PROGRAM OP10_ROBO
VAR
	I_OP10A_6000_6007						: BYTE_AS_BIT;	
	I_OP10A_6008_6015                       : BYTE_AS_BIT;
	I_OP10A_6016_6023                       : BYTE_AS_BIT;
	I_OP10A_6024_6031                       : BYTE_AS_BIT;
	I_OP10A_6032_6039                       : BYTE_AS_BIT;
	I_OP10A_6040_6047                       : BYTE_AS_BIT;
	I_OP10A_6048_6055                       : BYTE_AS_BIT;
	I_OP10A_6056_6063                       : BYTE_AS_BIT;
	O_OP10A_6000_6007						: BIT_AS_BYTE;
	O_OP10A_6008_6015						: BIT_AS_BYTE;
	O_OP10A_6016_6023						: BIT_AS_BYTE;
	O_OP10A_6024_6031						: BIT_AS_BYTE;
	O_OP10A_6032_6039						: BIT_AS_BYTE;
	O_OP10A_6040_6047						: BIT_AS_BYTE;
	O_OP10A_6048_6055						: BIT_AS_BYTE;
	O_OP10A_6056_6063						: BIT_AS_BYTE;

	I_OP10B_6000_6007						: BYTE_AS_BIT;	
	I_OP10B_6008_6015                       : BYTE_AS_BIT;
	I_OP10B_6016_6023                       : BYTE_AS_BIT;
	I_OP10B_6024_6031                       : BYTE_AS_BIT;
	I_OP10B_6032_6039                       : BYTE_AS_BIT;
	I_OP10B_6040_6047                       : BYTE_AS_BIT;
	I_OP10B_6048_6055                       : BYTE_AS_BIT;
	I_OP10B_6056_6063                       : BYTE_AS_BIT;
	O_OP10B_6032_6039						: BIT_AS_BYTE;
	O_OP10B_6040_6047						: BIT_AS_BYTE;
	O_OP10B_6048_6055						: BIT_AS_BYTE;
	O_OP10B_6056_6063						: BIT_AS_BYTE;
	O_OP10B_6000_6007						: BIT_AS_BYTE;
	O_OP10B_6008_6015						: BIT_AS_BYTE;
	O_OP10B_6016_6023						: BIT_AS_BYTE;
	O_OP10B_6024_6031						: BIT_AS_BYTE;

	OP10A_IP_ROBO_6000_6007  AT %I*			: USINT;
	OP10A_IP_ROBO_6008_6015  AT %I*			: USINT;
	OP10A_IP_ROBO_6016_6023  AT %I*			: USINT;
	OP10A_IP_ROBO_6024_6031  AT %I*			: USINT;
	OP10A_IP_ROBO_6032_6039  AT %I*			: USINT;
	OP10A_IP_ROBO_6040_6047  AT %I*			: USINT;	
	OP10A_IP_ROBO_6048_6055  AT %I*			: USINT;	
	OP10A_IP_ROBO_6056_6063  AT %I*			: USINT;	
	OP10A_OP_ROBO_6000_6007  AT %Q*			: USINT;
	OP10A_OP_ROBO_6008_6015  AT %Q*			: USINT;
	OP10A_OP_ROBO_6016_6023  AT %Q*			: USINT;
	OP10A_OP_ROBO_6024_6031  AT %Q*			: USINT;
	OP10A_OP_ROBO_6032_6039  AT %Q*			: USINT;
	OP10A_OP_ROBO_6040_6047  AT %Q*			: USINT;	
	OP10A_OP_ROBO_6048_6055  AT %Q*			: USINT;	
	OP10A_OP_ROBO_6056_6063  AT %Q*			: USINT;

	OP10B_IP_ROBO_6000_6007  AT %I*			: USINT;
	OP10B_IP_ROBO_6008_6015  AT %I*			: USINT;
	OP10B_IP_ROBO_6016_6023  AT %I*			: USINT;
	OP10B_IP_ROBO_6024_6031  AT %I*			: USINT;
	OP10B_IP_ROBO_6032_6039  AT %I*			: USINT;
	OP10B_IP_ROBO_6040_6047  AT %I*			: USINT;	
	OP10B_IP_ROBO_6048_6055  AT %I*			: USINT;	
	OP10B_IP_ROBO_6056_6063  AT %I*			: USINT;
	OP10B_OP_ROBO_6000_6007  AT %Q*			: USINT;
	OP10B_OP_ROBO_6008_6015  AT %Q*			: USINT;
	OP10B_OP_ROBO_6016_6023  AT %Q*			: USINT;
	OP10B_OP_ROBO_6024_6031  AT %Q*			: USINT;
	OP10B_OP_ROBO_6032_6039  AT %Q*			: USINT;
	OP10B_OP_ROBO_6040_6047  AT %Q*			: USINT;	
	OP10B_OP_ROBO_6048_6055  AT %Q*			: USINT;	
	OP10B_OP_ROBO_6056_6063  AT %Q*			: USINT;	


	


END_VAR

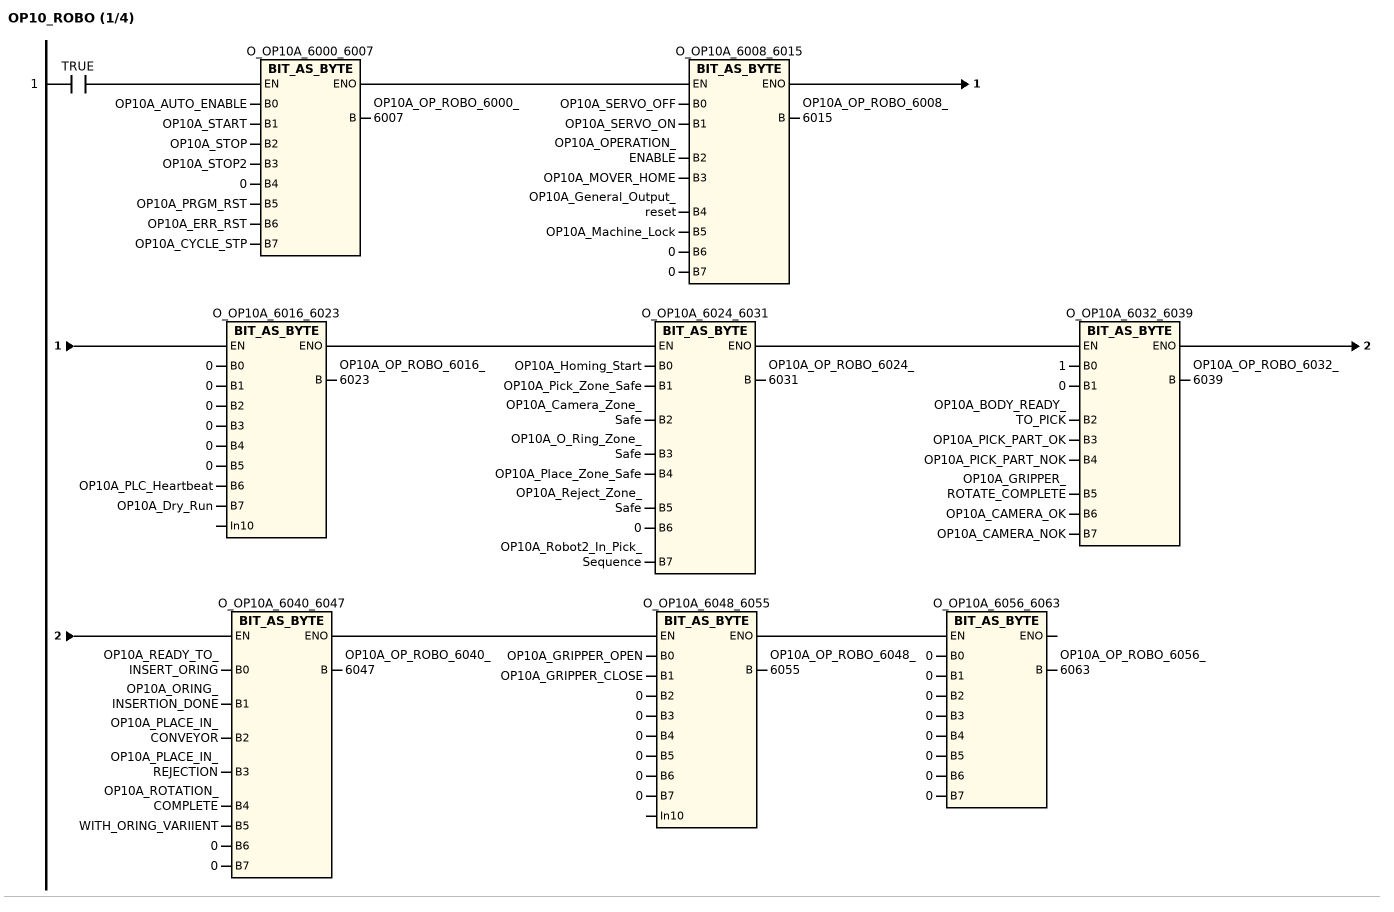
// NETWORK 1
O_OP10A_6000_6007(
    B0 := OP10A_AUTO_ENABLE,
    B1 := OP10A_START,
    B2 := OP10A_STOP,
    B3 := OP10A_STOP2,
    B4 := 0,
    B5 := OP10A_PRGM_RST,
    B6 := OP10A_ERR_RST,
    B7 := OP10A_CYCLE_STP,
    B => OP10A_OP_ROBO_6000_6007); // BIT_AS_BYTE
O_OP10A_6008_6015(
    B0 := OP10A_SERVO_OFF,
    B1 := OP10A_SERVO_ON,
    B2 := OP10A_OPERATION_ENABLE,
    B3 := OP10A_MOVER_HOME,
    B4 := OP10A_General_Output_reset,
    B5 := OP10A_Machine_Lock,
    B6 := 0,
    B7 := 0,
    B => OP10A_OP_ROBO_6008_6015); // BIT_AS_BYTE
O_OP10A_6016_6023(
    B0 := 0,
    B1 := 0,
    B2 := 0,
    B3 := 0,
    B4 := 0,
    B5 := 0,
    B6 := OP10A_PLC_Heartbeat,
    B7 := OP10A_Dry_Run,
    B => OP10A_OP_ROBO_6016_6023); // BIT_AS_BYTE
O_OP10A_6024_6031(
    B0 := OP10A_Homing_Start,
    B1 := OP10A_Pick_Zone_Safe,
    B2 := OP10A_Camera_Zone_Safe,
    B3 := OP10A_O_Ring_Zone_Safe,
    B4 := OP10A_Place_Zone_Safe,
    B5 := OP10A_Reject_Zone_Safe,
    B6 := 0,
    B7 := OP10A_Robot2_In_Pick_Sequence,
    B => OP10A_OP_ROBO_6024_6031); // BIT_AS_BYTE
O_OP10A_6032_6039(
    B0 := 1,
    B1 := 0,
    B2 := OP10A_BODY_READY_TO_PICK,
    B3 := OP10A_PICK_PART_OK,
    B4 := OP10A_PICK_PART_NOK,
    B5 := OP10A_GRIPPER_ROTATE_COMPLETE,
    B6 := OP10A_CAMERA_OK,
    B7 := OP10A_CAMERA_NOK,
    B => OP10A_OP_ROBO_6032_6039); // BIT_AS_BYTE
O_OP10A_6040_6047(
    B0 := OP10A_READY_TO_INSERT_ORING,
    B1 := OP10A_ORING_INSERTION_DONE,
    B2 := OP10A_PLACE_IN_CONVEYOR,
    B3 := OP10A_PLACE_IN_REJECTION,
    B4 := OP10A_ROTATION_COMPLETE,
    B5 := WITH_ORING_VARIIENT,
    B6 := 0,
    B7 := 0,
    B => OP10A_OP_ROBO_6040_6047); // BIT_AS_BYTE
O_OP10A_6048_6055(
    B0 := OP10A_GRIPPER_OPEN,
    B1 := OP10A_GRIPPER_CLOSE,
    B2 := 0,
    B3 := 0,
    B4 := 0,
    B5 := 0,
    B6 := 0,
    B7 := 0,
    B => OP10A_OP_ROBO_6048_6055); // BIT_AS_BYTE
O_OP10A_6056_6063(
    B0 := 0,
    B1 := 0,
    B2 := 0,
    B3 := 0,
    B4 := 0,
    B5 := 0,
    B6 := 0,
    B7 := 0,
    B => OP10A_OP_ROBO_6056_6063); // BIT_AS_BYTE

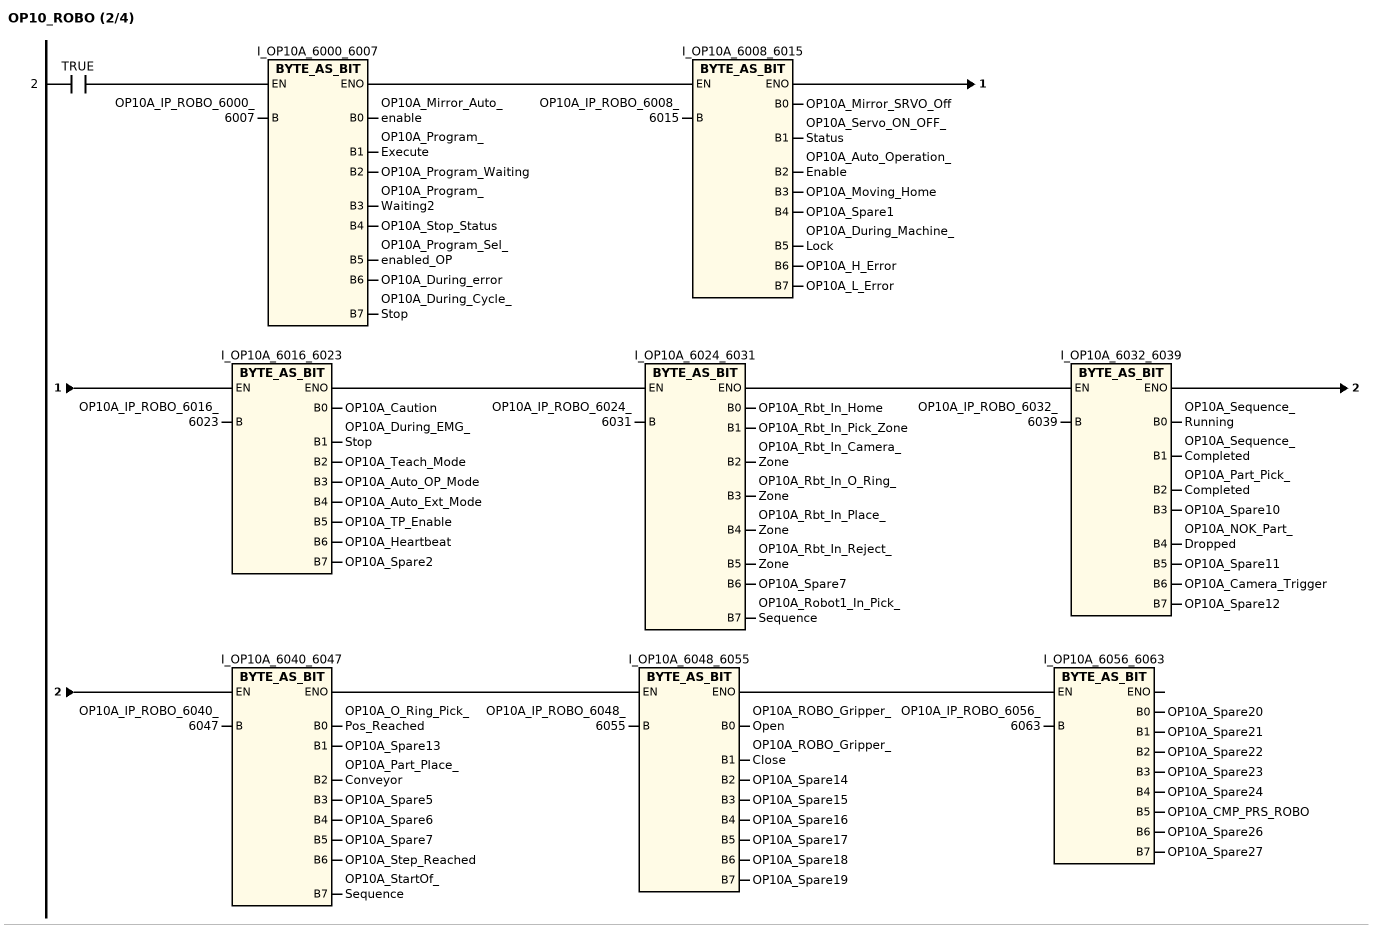
// NETWORK 2
I_OP10A_6000_6007(
    B := OP10A_IP_ROBO_6000_6007,
    B0 => OP10A_Mirror_Auto_enable,
    B1 => OP10A_Program_Execute,
    B2 => OP10A_Program_Waiting,
    B3 => OP10A_Program_Waiting2,
    B4 => OP10A_Stop_Status,
    B5 => OP10A_Program_Sel_enabled_OP,
    B6 => OP10A_During_error,
    B7 => OP10A_During_Cycle_Stop); // BYTE_AS_BIT
I_OP10A_6008_6015(
    B := OP10A_IP_ROBO_6008_6015,
    B0 => OP10A_Mirror_SRVO_Off,
    B1 => OP10A_Servo_ON_OFF_Status,
    B2 => OP10A_Auto_Operation_Enable,
    B3 => OP10A_Moving_Home,
    B4 => OP10A_Spare1,
    B5 => OP10A_During_Machine_Lock,
    B6 => OP10A_H_Error,
    B7 => OP10A_L_Error); // BYTE_AS_BIT
I_OP10A_6016_6023(
    B := OP10A_IP_ROBO_6016_6023,
    B0 => OP10A_Caution,
    B1 => OP10A_During_EMG_Stop,
    B2 => OP10A_Teach_Mode,
    B3 => OP10A_Auto_OP_Mode,
    B4 => OP10A_Auto_Ext_Mode,
    B5 => OP10A_TP_Enable,
    B6 => OP10A_Heartbeat,
    B7 => OP10A_Spare2); // BYTE_AS_BIT
I_OP10A_6024_6031(
    B := OP10A_IP_ROBO_6024_6031,
    B0 => OP10A_Rbt_In_Home,
    B1 => OP10A_Rbt_In_Pick_Zone,
    B2 => OP10A_Rbt_In_Camera_Zone,
    B3 => OP10A_Rbt_In_O_Ring_Zone,
    B4 => OP10A_Rbt_In_Place_Zone,
    B5 => OP10A_Rbt_In_Reject_Zone,
    B6 => OP10A_Spare7,
    B7 => OP10A_Robot1_In_Pick_Sequence); // BYTE_AS_BIT
I_OP10A_6032_6039(
    B := OP10A_IP_ROBO_6032_6039,
    B0 => OP10A_Sequence_Running,
    B1 => OP10A_Sequence_Completed,
    B2 => OP10A_Part_Pick_Completed,
    B3 => OP10A_Spare10,
    B4 => OP10A_NOK_Part_Dropped,
    B5 => OP10A_Spare11,
    B6 => OP10A_Camera_Trigger,
    B7 => OP10A_Spare12); // BYTE_AS_BIT
I_OP10A_6040_6047(
    B := OP10A_IP_ROBO_6040_6047,
    B0 => OP10A_O_Ring_Pick_Pos_Reached,
    B1 => OP10A_Spare13,
    B2 => OP10A_Part_Place_Conveyor,
    B3 => OP10A_Spare5,
    B4 => OP10A_Spare6,
    B5 => OP10A_Spare7,
    B6 => OP10A_Step_Reached,
    B7 => OP10A_StartOf_Sequence); // BYTE_AS_BIT
I_OP10A_6048_6055(
    B := OP10A_IP_ROBO_6048_6055,
    B0 => OP10A_ROBO_Gripper_Open,
    B1 => OP10A_ROBO_Gripper_Close,
    B2 => OP10A_Spare14,
    B3 => OP10A_Spare15,
    B4 => OP10A_Spare16,
    B5 => OP10A_Spare17,
    B6 => OP10A_Spare18,
    B7 => OP10A_Spare19); // BYTE_AS_BIT
I_OP10A_6056_6063(
    B := OP10A_IP_ROBO_6056_6063,
    B0 => OP10A_Spare20,
    B1 => OP10A_Spare21,
    B2 => OP10A_Spare22,
    B3 => OP10A_Spare23,
    B4 => OP10A_Spare24,
    B5 => OP10A_CMP_PRS_ROBO,
    B6 => OP10A_Spare26,
    B7 => OP10A_Spare27); // BYTE_AS_BIT

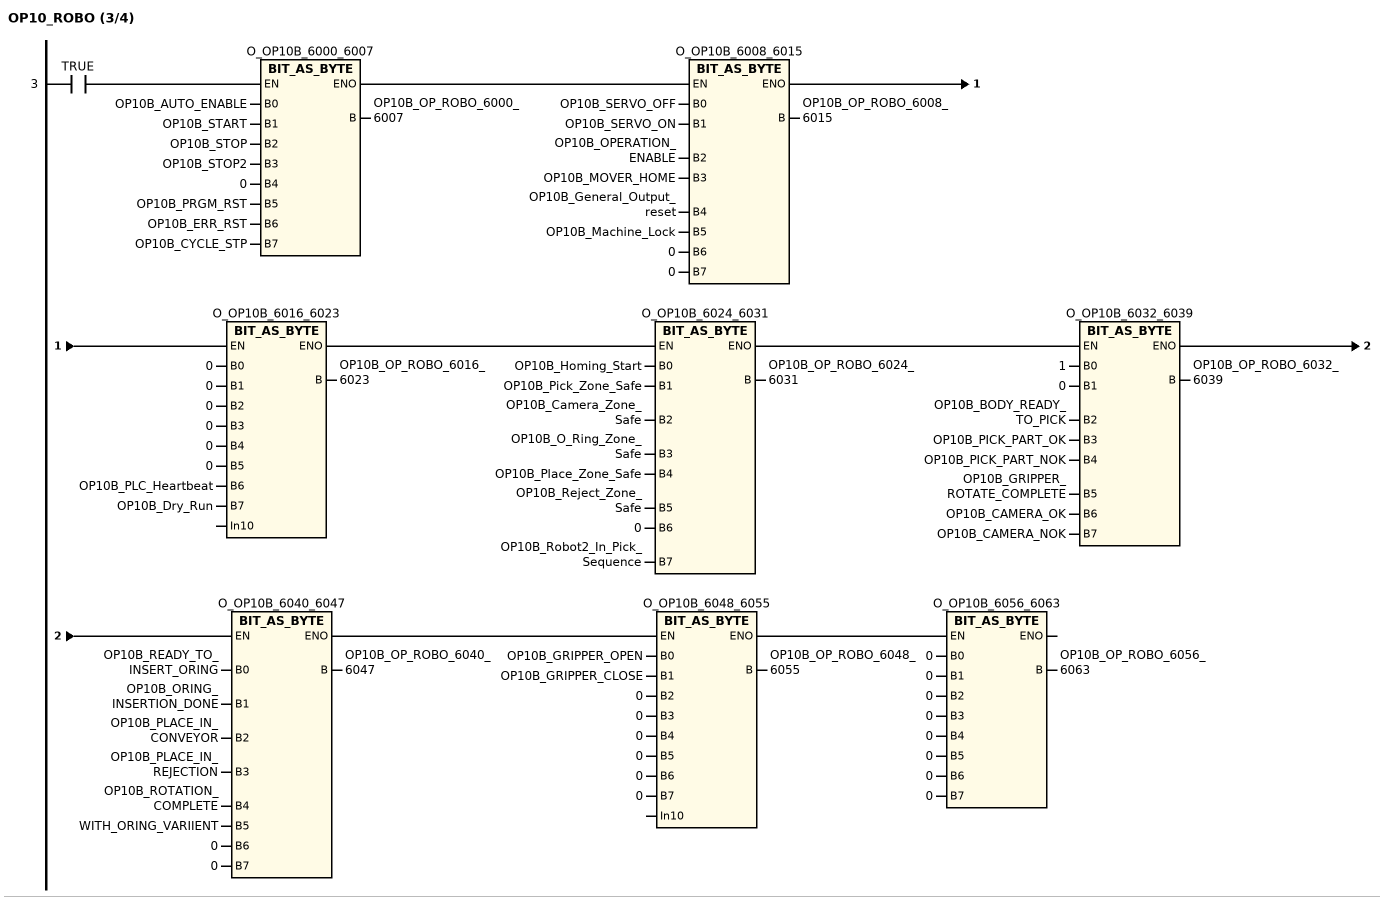
// NETWORK 3
O_OP10B_6000_6007(
    B0 := OP10B_AUTO_ENABLE,
    B1 := OP10B_START,
    B2 := OP10B_STOP,
    B3 := OP10B_STOP2,
    B4 := 0,
    B5 := OP10B_PRGM_RST,
    B6 := OP10B_ERR_RST,
    B7 := OP10B_CYCLE_STP,
    B => OP10B_OP_ROBO_6000_6007); // BIT_AS_BYTE
O_OP10B_6008_6015(
    B0 := OP10B_SERVO_OFF,
    B1 := OP10B_SERVO_ON,
    B2 := OP10B_OPERATION_ENABLE,
    B3 := OP10B_MOVER_HOME,
    B4 := OP10B_General_Output_reset,
    B5 := OP10B_Machine_Lock,
    B6 := 0,
    B7 := 0,
    B => OP10B_OP_ROBO_6008_6015); // BIT_AS_BYTE
O_OP10B_6016_6023(
    B0 := 0,
    B1 := 0,
    B2 := 0,
    B3 := 0,
    B4 := 0,
    B5 := 0,
    B6 := OP10B_PLC_Heartbeat,
    B7 := OP10B_Dry_Run,
    B => OP10B_OP_ROBO_6016_6023); // BIT_AS_BYTE
O_OP10B_6024_6031(
    B0 := OP10B_Homing_Start,
    B1 := OP10B_Pick_Zone_Safe,
    B2 := OP10B_Camera_Zone_Safe,
    B3 := OP10B_O_Ring_Zone_Safe,
    B4 := OP10B_Place_Zone_Safe,
    B5 := OP10B_Reject_Zone_Safe,
    B6 := 0,
    B7 := OP10B_Robot2_In_Pick_Sequence,
    B => OP10B_OP_ROBO_6024_6031); // BIT_AS_BYTE
O_OP10B_6032_6039(
    B0 := 1,
    B1 := 0,
    B2 := OP10B_BODY_READY_TO_PICK,
    B3 := OP10B_PICK_PART_OK,
    B4 := OP10B_PICK_PART_NOK,
    B5 := OP10B_GRIPPER_ROTATE_COMPLETE,
    B6 := OP10B_CAMERA_OK,
    B7 := OP10B_CAMERA_NOK,
    B => OP10B_OP_ROBO_6032_6039); // BIT_AS_BYTE
O_OP10B_6040_6047(
    B0 := OP10B_READY_TO_INSERT_ORING,
    B1 := OP10B_ORING_INSERTION_DONE,
    B2 := OP10B_PLACE_IN_CONVEYOR,
    B3 := OP10B_PLACE_IN_REJECTION,
    B4 := OP10B_ROTATION_COMPLETE,
    B5 := WITH_ORING_VARIIENT,
    B6 := 0,
    B7 := 0,
    B => OP10B_OP_ROBO_6040_6047); // BIT_AS_BYTE
O_OP10B_6048_6055(
    B0 := OP10B_GRIPPER_OPEN,
    B1 := OP10B_GRIPPER_CLOSE,
    B2 := 0,
    B3 := 0,
    B4 := 0,
    B5 := 0,
    B6 := 0,
    B7 := 0,
    B => OP10B_OP_ROBO_6048_6055); // BIT_AS_BYTE
O_OP10B_6056_6063(
    B0 := 0,
    B1 := 0,
    B2 := 0,
    B3 := 0,
    B4 := 0,
    B5 := 0,
    B6 := 0,
    B7 := 0,
    B => OP10B_OP_ROBO_6056_6063); // BIT_AS_BYTE

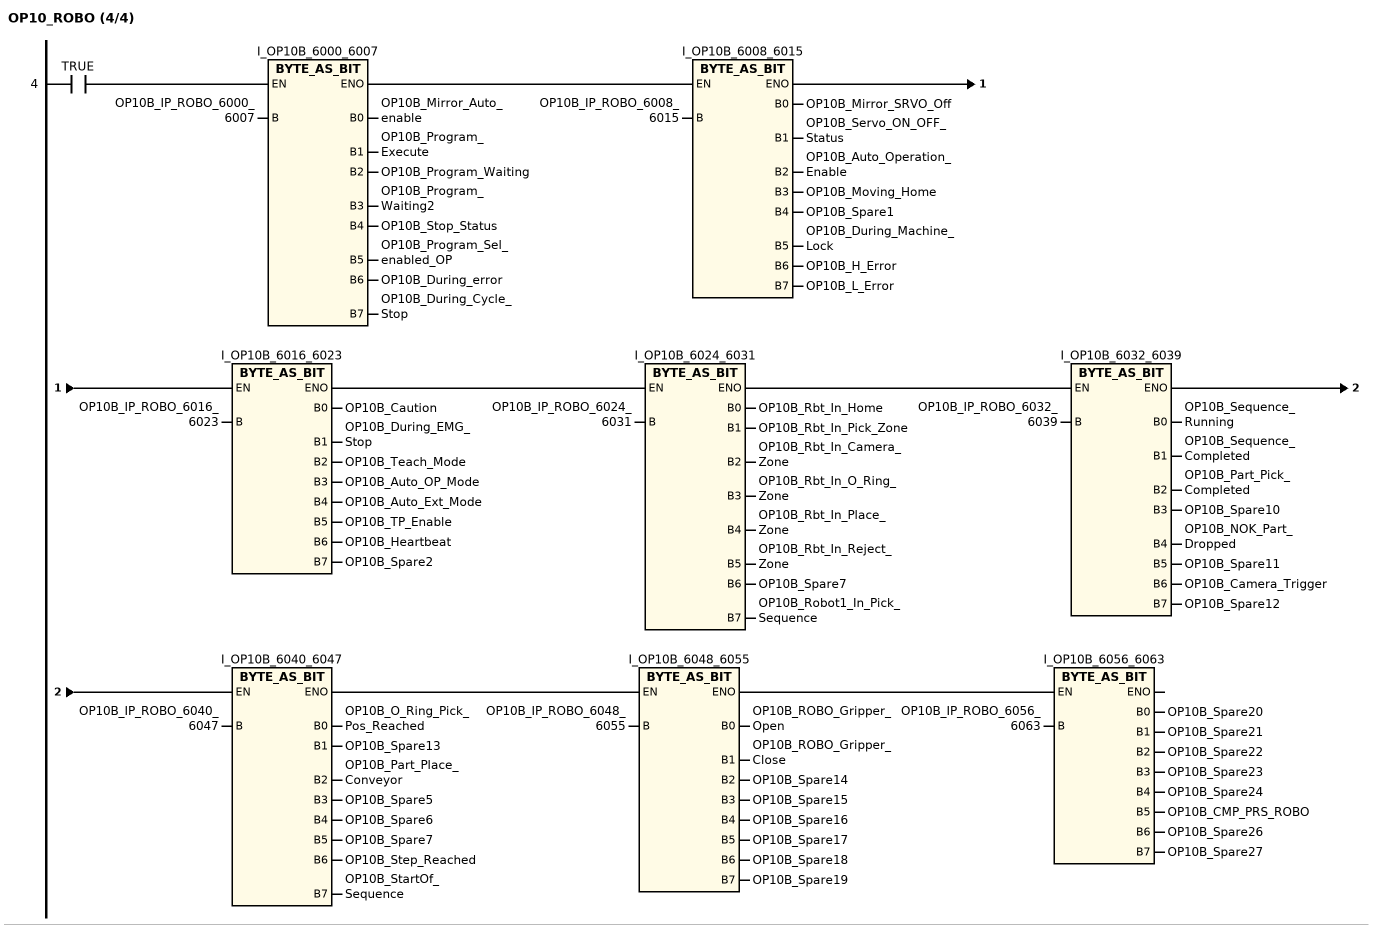
// NETWORK 4
I_OP10B_6000_6007(
    B := OP10B_IP_ROBO_6000_6007,
    B0 => OP10B_Mirror_Auto_enable,
    B1 => OP10B_Program_Execute,
    B2 => OP10B_Program_Waiting,
    B3 => OP10B_Program_Waiting2,
    B4 => OP10B_Stop_Status,
    B5 => OP10B_Program_Sel_enabled_OP,
    B6 => OP10B_During_error,
    B7 => OP10B_During_Cycle_Stop); // BYTE_AS_BIT
I_OP10B_6008_6015(
    B := OP10B_IP_ROBO_6008_6015,
    B0 => OP10B_Mirror_SRVO_Off,
    B1 => OP10B_Servo_ON_OFF_Status,
    B2 => OP10B_Auto_Operation_Enable,
    B3 => OP10B_Moving_Home,
    B4 => OP10B_Spare1,
    B5 => OP10B_During_Machine_Lock,
    B6 => OP10B_H_Error,
    B7 => OP10B_L_Error); // BYTE_AS_BIT
I_OP10B_6016_6023(
    B := OP10B_IP_ROBO_6016_6023,
    B0 => OP10B_Caution,
    B1 => OP10B_During_EMG_Stop,
    B2 => OP10B_Teach_Mode,
    B3 => OP10B_Auto_OP_Mode,
    B4 => OP10B_Auto_Ext_Mode,
    B5 => OP10B_TP_Enable,
    B6 => OP10B_Heartbeat,
    B7 => OP10B_Spare2); // BYTE_AS_BIT
I_OP10B_6024_6031(
    B := OP10B_IP_ROBO_6024_6031,
    B0 => OP10B_Rbt_In_Home,
    B1 => OP10B_Rbt_In_Pick_Zone,
    B2 => OP10B_Rbt_In_Camera_Zone,
    B3 => OP10B_Rbt_In_O_Ring_Zone,
    B4 => OP10B_Rbt_In_Place_Zone,
    B5 => OP10B_Rbt_In_Reject_Zone,
    B6 => OP10B_Spare7,
    B7 => OP10B_Robot1_In_Pick_Sequence); // BYTE_AS_BIT
I_OP10B_6032_6039(
    B := OP10B_IP_ROBO_6032_6039,
    B0 => OP10B_Sequence_Running,
    B1 => OP10B_Sequence_Completed,
    B2 => OP10B_Part_Pick_Completed,
    B3 => OP10B_Spare10,
    B4 => OP10B_NOK_Part_Dropped,
    B5 => OP10B_Spare11,
    B6 => OP10B_Camera_Trigger,
    B7 => OP10B_Spare12); // BYTE_AS_BIT
I_OP10B_6040_6047(
    B := OP10B_IP_ROBO_6040_6047,
    B0 => OP10B_O_Ring_Pick_Pos_Reached,
    B1 => OP10B_Spare13,
    B2 => OP10B_Part_Place_Conveyor,
    B3 => OP10B_Spare5,
    B4 => OP10B_Spare6,
    B5 => OP10B_Spare7,
    B6 => OP10B_Step_Reached,
    B7 => OP10B_StartOf_Sequence); // BYTE_AS_BIT
I_OP10B_6048_6055(
    B := OP10B_IP_ROBO_6048_6055,
    B0 => OP10B_ROBO_Gripper_Open,
    B1 => OP10B_ROBO_Gripper_Close,
    B2 => OP10B_Spare14,
    B3 => OP10B_Spare15,
    B4 => OP10B_Spare16,
    B5 => OP10B_Spare17,
    B6 => OP10B_Spare18,
    B7 => OP10B_Spare19); // BYTE_AS_BIT
I_OP10B_6056_6063(
    B := OP10B_IP_ROBO_6056_6063,
    B0 => OP10B_Spare20,
    B1 => OP10B_Spare21,
    B2 => OP10B_Spare22,
    B3 => OP10B_Spare23,
    B4 => OP10B_Spare24,
    B5 => OP10B_CMP_PRS_ROBO,
    B6 => OP10B_Spare26,
    B7 => OP10B_Spare27); // BYTE_AS_BIT

END_PROGRAM

(* stored: Version 1.1.0.1, ProductVersion 3.1.4024.11
   POU OP10_ROBO: Id {101dcb0a-72d9-4e84-b25a-1b99a60cd138}, SpecialFunc None *)
